PROGRAM TORCHCLEAN
VAR_INPUT
	KR_TC	: BOOL;
	process_A	: INT;
END_VAR
VAR
	TC_sequence	: INT;
END_VAR


CASE TC_sequence OF
	0:
		IF process_A = 0 THEN
			IF KR1.Idle AND KR2.Idle AND KR3.Idle AND KR4.Idle THEN
				KR3.bOutBit[3,2]:= TRUE; //302
				KR4.bOutBit[3,1] := TRUE; //301
				KR_TC := TRUE;
				process_A := 1;
				RETURN;
			END_IF
		ELSIF process_A = 1 THEN
			IF KR3.bInBit[3,2] AND KR4.bInBit[3,1] THEN
				KR3.bOutBit[3,2]:= FALSE; //302
				KR4.bOutBit[3,1] := FALSE; //301
				process_A := 2;
				RETURN;
			END_IF	
		ELSIF process_A = 2 THEN
			IF NOT KR3.bInBit[3,2] AND NOT KR4.bInBit[3,1] THEN
				process_A:= 3;
				RETURN;
			END_IF	
		ELSIF process_A = 3 THEN
			IF KR3.Idle AND KR4.Idle THEN
				KR_TC := FALSE;
				MAIN.btnTorchClean := FALSE;
				process_A := 0;
				TC_sequence := 0;
			END_IF
		END_IF
END_CASE

END_PROGRAM

(* stored: Version 1.1.0.1, ProductVersion 3.1.4024.12
   POU TORCHCLEAN: Id {8e0b119b-a45e-4f6a-9750-8aa306d1c175}, SpecialFunc None *)
